PROGRAM MAIN
VAR
END_VAR

END_PROGRAM

(* stored: Version 1.1.0.1
   POU MAIN: Id {6936711f-aee1-47f6-8b72-e1a06991e1fe} *)
